FUNCTION_BLOCK Door_HMI (* Service Interface Function Block Type *)
  (* Standard: 61499-2 *)
  (* Version 0.0, 6/3/2016, Andrei, nxtControl GmbH, template *)
  PACKAGE Main;
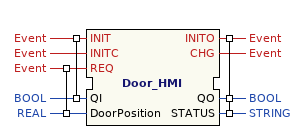
  EVENT_INPUT
    INIT WITH QI;
    INITC;
    REQ WITH DoorPosition;
  END_EVENT
  EVENT_OUTPUT
    INITO WITH QO, STATUS;
    CHG;
  END_EVENT
  VAR_INPUT
    QI : BOOL;
    DoorPosition : REAL;
  END_VAR
  VAR_OUTPUT
    QO : BOOL; (* Event Output Qualifier *)
    STATUS : STRING; (* Service Status *)
  END_VAR
END_FUNCTION_BLOCK
